Fanuc KAREL source: kc00032.KL

PROGRAM KC00032
%STACKSIZE=65535
%PRIORITY=65535
%NOLOCKGROUP
VAR
I : INTEGER
J : INTEGER
K : INTEGER
R : REAL
B : BOOLEAN
S : STRING[80]
T : STRING[80]
AI : ARRAY[8] OF INTEGER
AB : ARRAY[244] OF BYTE
SA : ARRAY[8] OF STRING[80]
-- UNRESOLVED DECLARATIONS (source type spelling not recovered)
-- P : TYPE_0x001F (type_u16=0x001F)
-- Q : TYPE_0x001F (type_u16=0x001F)
BEGIN
PROG_LIST(S,I,J,K,SA,I,J,1)
END KC00032
